PROGRAM POU_Parada
VAR
END_VAR

GVL.Emitter_1:= FALSE;
//Semáforo indicando estación que se ha solicitado su parada
GVL.Stack_Light_1_Green := FALSE;
GVL.Stack_Light_1_Red := FALSE;	
GVL.Stack_Light_1_Yellow := TRUE;

GVL.Factory_IO_Pause := TRUE;

END_PROGRAM

(* stored: Version 1.1.0.1, ProductVersion 3.1.4024.12
   POU POU_Parada: Id {4fbb0307-13ef-431c-9f14-d054c15cba7d}, SpecialFunc None *)
